# EPICS IOC start-up script: iocBoot/iocoh26/iocsh/motors.iocsh
# ANG1 motors Command file Example
#
### Note:  Modbus support (the EPICS modbus module) is required to be included in the
###        EPICS application where the ANG1 support will be loaded.  This file is an
###        example of how to load the ANG1 support, in an ioc that is built with the
###        EPICS modbus module.

# Use the following commands for TCP/IP
#drvAsynIPPortConfigure(const char *portName,
#                       const char *hostInfo,
#                       unsigned int priority,
#                       int noAutoConnect,
#                       int noProcessEos);
# One per controller.  One controller can support up to six drivers.
drvAsynIPPortConfigure("ang1_1","192.168.100.21:502",0,0,1)
#drvAsynIPPortConfigure("ang1_2","192.168.1.32:502",0,0,1)
#drvAsynIPPortConfigure("ang1_3","192.168.xxx.xxx:502",0,0,1)

#modbusInterposeConfig(const char *portName,
#                      modbusLinkType linkType,
#                      int timeoutMsec,
#                      int writeDelayMsec)
# One per controller.  One controller can support up to six drivers.
modbusInterposeConfig("ang1_1",0,2000,0)
#modbusInterposeConfig("ang1_2",0,2000,0)

# Word access at Modbus address 0
# Access 1 words as inputs.
# Function code=3
# default data type unsigned integer.
# drvModbusAsynConfigure("portName", "tcpPortName", slaveAddress, modbusFunction, modbusStartAddress, modbusLength, dataType, pollMsec, "plcType")
# One per axis.  Note: "ANG1" is the AMCI model. "ANG1_1" is the controller.  "ANG1_1_1" is the axis.
drvModbusAsynConfigure("ANG1_1_1_In_Word", "ang1_1", 0, 4, 0,  10, 0, 100, "ANG1_stepper")
# drvModbusAsynConfigure("ANG1_1_2_In_Word", "ang1_1", 0, 4, 10, 10, 0, 100, "ANG1_stepper")
#drvModbusAsynConfigure("ANG1_1_3_In_Word", "ang1_1", 0, 3, 20, 10, 0, 100, "ANG1_stepper")
#drvModbusAsynConfigure("ANG1_1_4_In_Word", "ang1_1", 0, 3, 30, 10, 0, 100, "ANG1_stepper")
#drvModbusAsynConfigure("ANG1_1_5_In_Word", "ang1_1", 0, 3, 40, 10, 0, 100, "ANG1_stepper")
#drvModbusAsynConfigure("ANG1_1_6_In_Word", "ang1_1", 0, 3, 50, 10, 0, 100, "ANG1_stepper")

# Access 1 words as outputs.
# Either function code=6 (single register) or 16 (multiple registers) can be used, but 16
# is better because it is "atomic" when writing values longer than 16-bits.
# Default data type unsigned integer.
# drvModbusAsynConfigure("portName", "tcpPortName", slaveAddress, modbusFunction, modbusStartAddress, modbusLength, dataType, pollMsec, "plcType")
# Not sure why the outputs can't be configured for Modbus data type 4?
drvModbusAsynConfigure("ANG1_1_1_Out_Word", "ang1_1", 0, 6, 1024, 10, 0, 1, "ANG1_stepper")
# drvModbusAsynConfigure("ANG1_1_2_Out_Word", "ang1_1", 0, 6, 1034, 10, 0, 1, "ANG1_stepper")
#drvModbusAsynConfigure("ANG1_1_3_Out_Word", "ang1_1", 0, 6, 1044, 10, 0, 1, "ANG1_stepper")
#drvModbusAsynConfigure("ANG1_1_4_Out_Word", "ang1_1", 0, 6, 1054, 10, 0, 1, "ANG1_stepper")
#drvModbusAsynConfigure("ANG1_1_5_Out_Word", "ang1_1", 0, 6, 1064, 10, 0, 1, "ANG1_stepper")
#drvModbusAsynConfigure("ANG1_1_6_Out_Word", "ang1_1", 0, 6, 1074, 10, 0, 1, "ANG1_stepper")

# Second ANG1 controller...
#drvModbusAsynConfigure("ANG1_2_1_Out_Word_0", "ang1_2", 0, 6, 1024, 1, 0, 1, "ANG1_stepper")

dbLoadTemplate("substitutions/motor.substitutions", "P=$(PREFIX)")

# AMCI ANG1 stepper controller/driver support
#  portName  		The name of the asyn port that will be created for this driver
#  ANG1InPortName  	The name of the In drvAsynIPPPort that was created previously to connect to the ANG1 controller
#  ANG1OutPortName  The name of the Out drvAsynIPPPort that was created previously to connect to the ANG1 controller
#  numAxes			The number of axes that this controller supports
#  movingPollPeriod The time in ms between polls when any axis is moving
#  idlePollPeriod	The time in ms between polls when no axis is moving
#
# One per axis.  Note: "ANG1" is the AMCI model. "ANG1_1" is the controller.  "ANG1_1_1" is the axis.
# Also, ANG1_1_1 is the port name needed for motor.substitutions.
ANG1CreateController(ANG1_1_1, ANG1_1_1_In_Word, ANG1_1_1_Out_Word, 1, 100, 0)
# ANG1CreateController(ANG1_1_2, ANG1_1_2_In_Word, ANG1_1_2_Out_Word, 1, 100, 0)
#ANG1CreateController(ANG1_1, ANG1_1_3_In_Word, ANG1_1_3_Out_Word, 1, 100, 0)
#ANG1CreateController(ANG1_1, ANG1_1_4_In_Word, ANG1_1_4_Out_Word, 1, 100, 0)
#ANG1CreateController(ANG1_1, ANG1_1_5_In_Word, ANG1_1_5_Out_Word, 1, 100, 0)
#ANG1CreateController(ANG1_1, ANG1_1_6_In_Word, ANG1_1_6_Out_Word, 1, 100, 0)

# Load scan stuff for this motor
dbLoadRecords("$(SSCAN)/sscanApp/Db/scanParms.db", "P=$(PREFIX),SCANREC=$(PREFIX)scan1,Q=m1,POS=m1.VAL,RDBK=m1.RBV")

# allstop, alldone
iocshLoad("$(MOTOR)/iocsh/allstop.iocsh", "P=$(PREFIX)")
